(* IEC 61131-3 sources: test/Class/HmiColorMap, 1 file *)

(* ---- HmiColorMap.st ---- *)
(*!
<Class
	Name               = "HmiColorMap"
	Revision           = "0.0"
	RealtimeTask       = "false"
	CyclicTask         = "false"
	BackgroundTask     = "false"
	Sigmatek           = "true"
	OSInterface        = "false"
	HighPriority       = "false"
	Automatic          = "false"
	UpdateMode         = "Prescan"
	SharedCommandTable = "true"
	Objectsize         = "(284,120)">
	<Channels>
	</Channels>
	<Network Name="HmiColorMap">
		<!-- List of Components in this network -->
		<Components>
			<Object
				Name       = "_base"
				Class      = "HmiBaseList"
				Position   = "(218,120)"
				Visualized = "false">
				<Channels>
					<Server Name="ClassSvr"/>
					<Client Name="File"/>
				</Channels>
			</Object>
		</Components>
		<Comments>
		</Comments>
		<!-- List of Connections in this network -->
		<Connections>
			<Connection Source="this.ClassSvr" Destination="_base.ClassSvr" Vertices="(690,210),(518,210),"/>
			<Connection Source="_base.File" Destination="this.File" Vertices="(218,210),(38,210),"/>
		</Connections>
		<!-- Headerfiles -->
		<Options>
		</Options>
	</Network>
</Class>
*)
#pragma using HmiBaseList

HmiColorMap : CLASS
: HmiBaseList
  //Servers:
  //Clients:
  //Variables:
		Ptr : ARRAY [0..255] OF UINT;

		No 	: UDINT;
  //Functions:

	FUNCTION HmiColorMap
		VAR_OUTPUT
			ret_code 	: ConfStates;
		END_VAR;

	FUNCTION VIRTUAL Load
		VAR_OUTPUT
			retcode 	: BOOL;
		END_VAR;

	FUNCTION VIRTUAL Free;

	FUNCTION GLOBAL Get
		VAR_INPUT
			index 	: USINT;
		END_VAR
		VAR_OUTPUT
			retcode 	: UINT;
		END_VAR;
  //Tables:
	FUNCTION @STD
		VAR_OUTPUT
			ret_code	: CONFSTATES;
		END_VAR;
	FUNCTION GLOBAL TAB @CT_;
END_CLASS;

FUNCTION HmiColorMap::HmiColorMap
	VAR_OUTPUT
		ret_code 	: ConfStates;
	END_VAR

	ret_code := C_OK;
  No := 0;

END_FUNCTION

FUNCTION MakeCol16 VAR_INPUT cr : UINT; cg : UINT; cb : UINT; END_VAR
	VAR_OUTPUT
		retcode 	: UINT;
	END_VAR

  if(cb = 254) then
    if((cr = 255) & (cg = 255)) then
      retcode := 0xFFFE;  // transparent
      return;
    end_if;
  end_if;

  cr      := (cr and 16#F8);
  cg      := (cg and 16#FC);
  cb      := (cb and 16#F8);
  retcode := (cr shl 8) or (cg shl 3) or (cb shr 3);

END_FUNCTION

FUNCTION VIRTUAL HmiColorMap::Free

  No := 0;

END_FUNCTION

FUNCTION VIRTUAL HmiColorMap::Load
	VAR_OUTPUT
		retcode 	: BOOL;
	END_VAR
  VAR
    rgb : array[0..2] of usint;
  	anz : udint;
    ph : ^uint;
  END_VAR

  retcode := false;
  File.Fread(#anz, 4);
  if(anz = 256) then

    ph := #Ptr[0];
    while(anz) do
      anz -= 1;
      File.FRead(#rgb[0], 3);
      ph^ := MakeCol16(rgb[0], rgb[1], rgb[2]);

      ph  += 2;
    end_while;

    retcode := File.FChkFile();
    No := 256;
  end_if;

  if(retcode = true) then
    ClassSvr := to_dint(No);
  end_if;

END_FUNCTION

FUNCTION GLOBAL HmiColorMap::Get
	VAR_INPUT
		index 	: USINT;
	END_VAR
	VAR_OUTPUT
		retcode 	: UINT;
	END_VAR

  retcode := 16#FFFF;
  if(index < No) then
    retcode := Ptr[index];
  end_if;

END_FUNCTION
